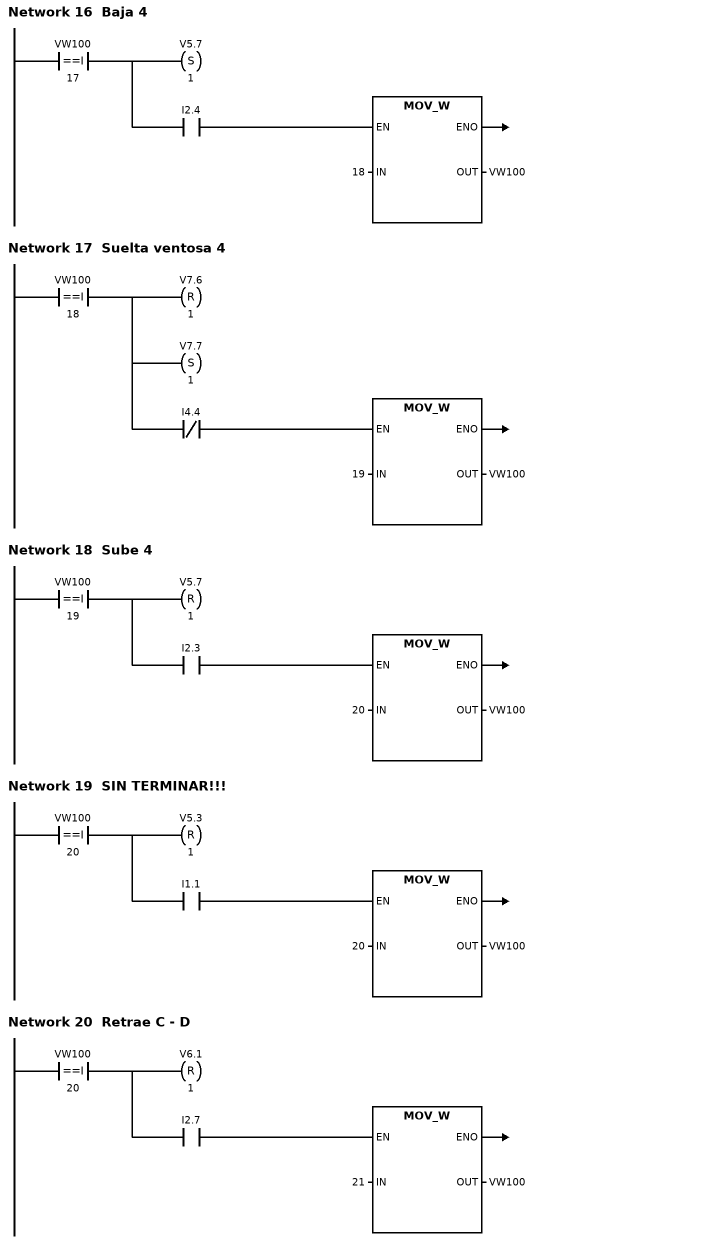
[picture p24: SBR1 networks 16-20]
Network 16 // Baja 4
LDW=   VW100, 17
S      V5.7, 1
A      I2.4
MOVW   18, VW100
Network 17 // Suelta ventosa 4
LDW=   VW100, 18
R      V7.6, 1
S      V7.7, 1
AN     I4.4
MOVW   19, VW100
Network 18 // Sube 4
LDW=   VW100, 19
R      V5.7, 1
A      I2.3
MOVW   20, VW100
Network 19 // SIN TERMINAR!!!
LDW=   VW100, 20
R      V5.3, 1
A      I1.1
MOVW   20, VW100
Network 20 // Retrae C - D
LDW=   VW100, 20
R      V6.1, 1
A      I2.7
MOVW   21, VW100
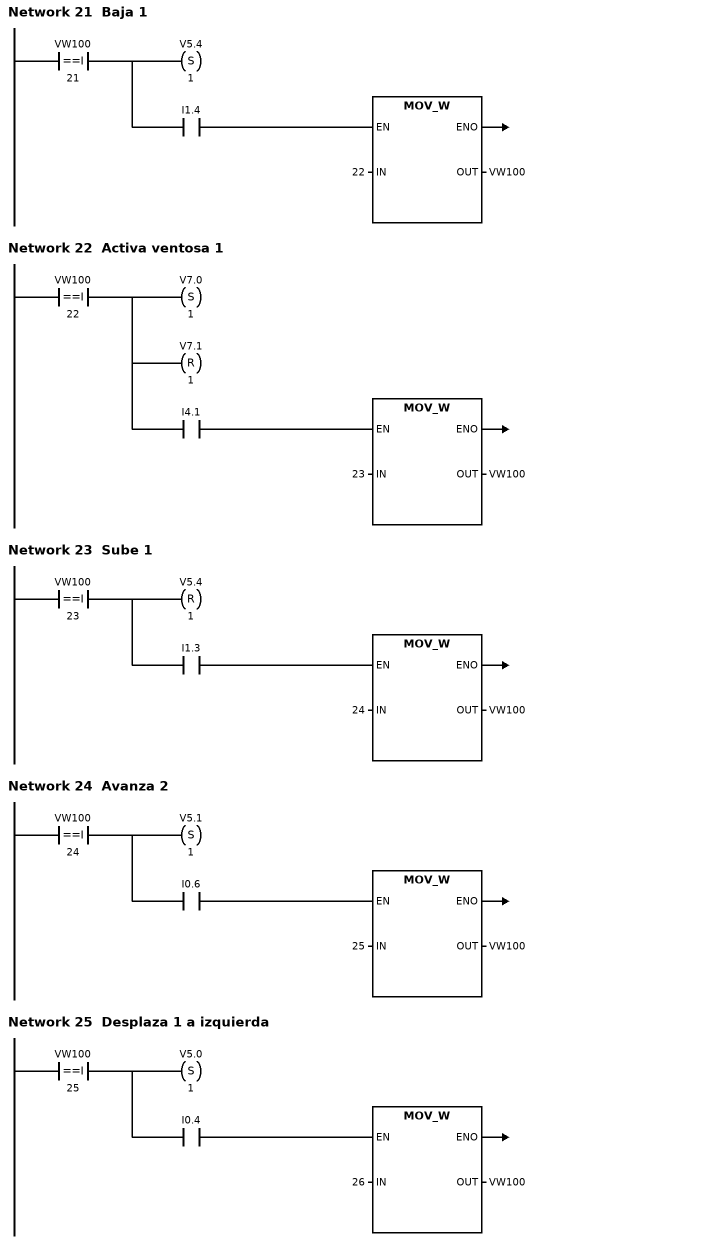
Network 21 // Baja 1
LDW=   VW100, 21
S      V5.4, 1
A      I1.4
MOVW   22, VW100
Network 22 // Activa ventosa 1
LDW=   VW100, 22
S      V7.0, 1
R      V7.1, 1
A      I4.1
MOVW   23, VW100
Network 23 // Sube 1
LDW=   VW100, 23
R      V5.4, 1
A      I1.3
MOVW   24, VW100
Network 24 // Avanza 2
LDW=   VW100, 24
S      V5.1, 1
A      I0.6
MOVW   25, VW100
Network 25 // Desplaza 1 a izquierda
LDW=   VW100, 25
S      V5.0, 1
A      I0.4
MOVW   26, VW100
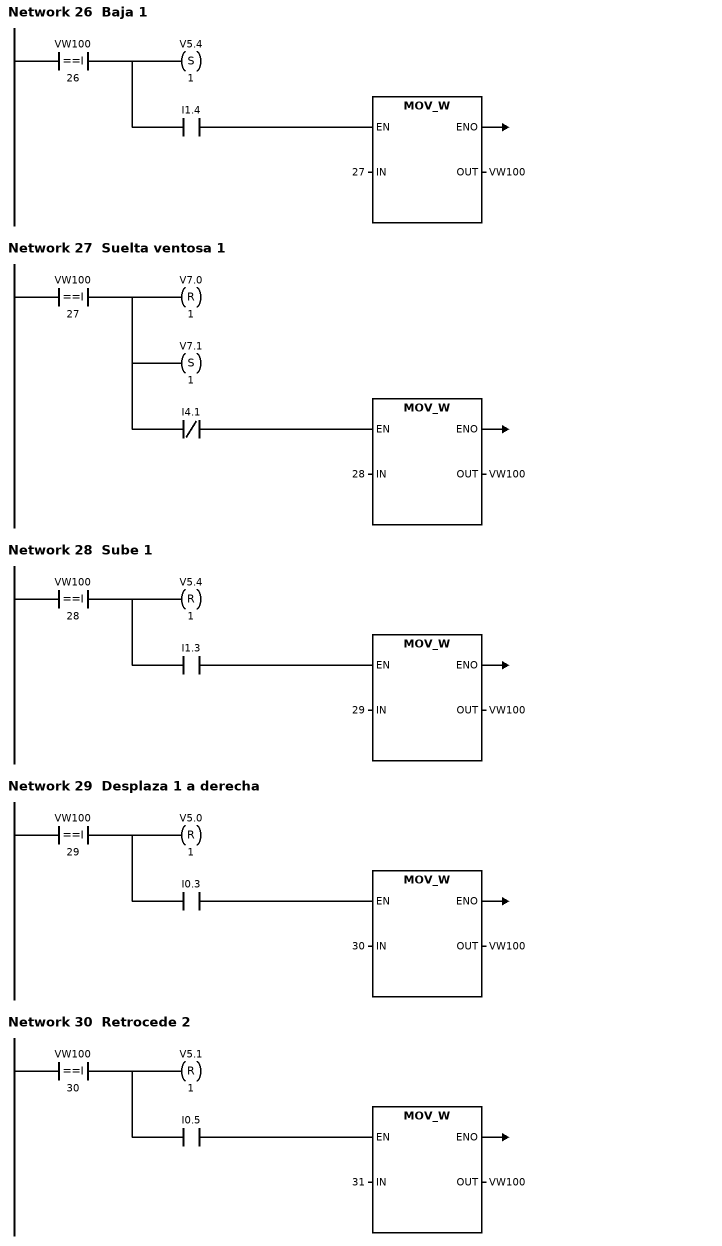
Network 26 // Baja 1
LDW=   VW100, 26
S      V5.4, 1
A      I1.4
MOVW   27, VW100
Network 27 // Suelta ventosa 1
LDW=   VW100, 27
R      V7.0, 1
S      V7.1, 1
AN     I4.1
MOVW   28, VW100
Network 28 // Sube 1
LDW=   VW100, 28
R      V5.4, 1
A      I1.3
MOVW   29, VW100
Network 29 // Desplaza 1 a derecha
LDW=   VW100, 29
R      V5.0, 1
A      I0.3
MOVW   30, VW100
Network 30 // Retrocede 2
LDW=   VW100, 30
R      V5.1, 1
A      I0.5
MOVW   31, VW100
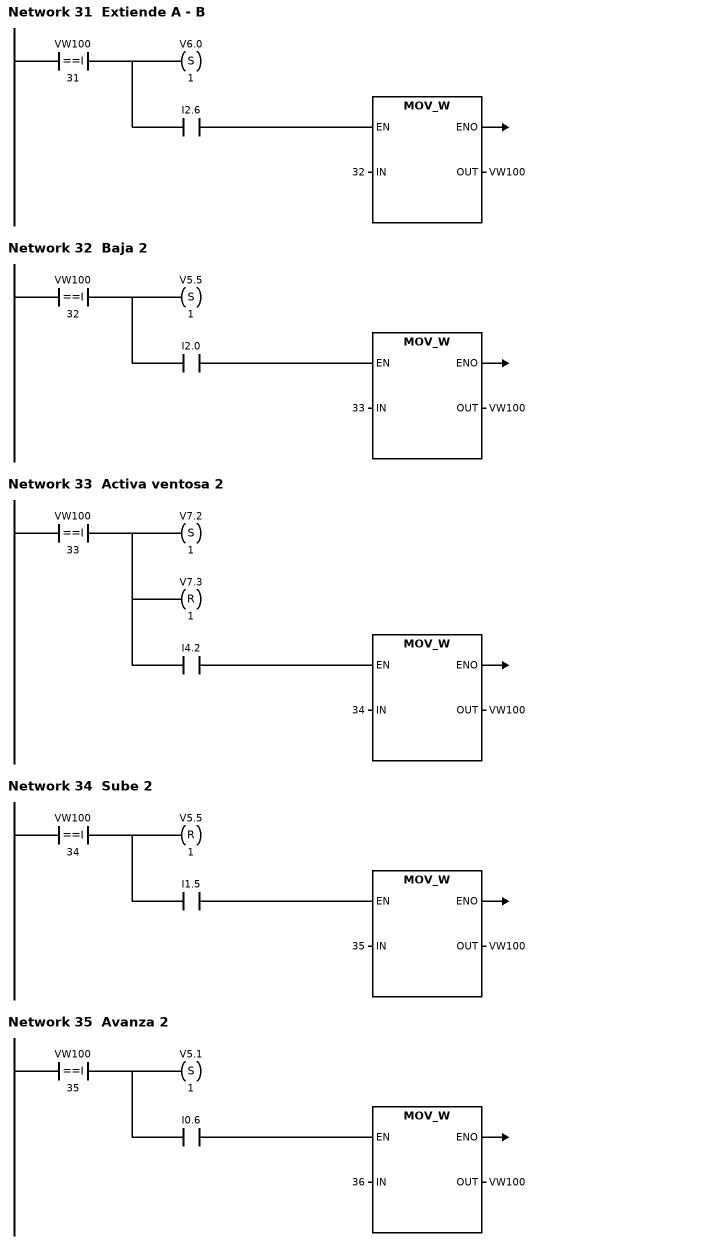
Network 31 // Extiende A - B
LDW=   VW100, 31
S      V6.0, 1
A      I2.6
MOVW   32, VW100
Network 32 // Baja 2
LDW=   VW100, 32
S      V5.5, 1
A      I2.0
MOVW   33, VW100
Network 33 // Activa ventosa 2
LDW=   VW100, 33
S      V7.2, 1
R      V7.3, 1
A      I4.2
MOVW   34, VW100
Network 34 // Sube 2
LDW=   VW100, 34
R      V5.5, 1
A      I1.5
MOVW   35, VW100
Network 35 // Avanza 2
LDW=   VW100, 35
S      V5.1, 1
A      I0.6
MOVW   36, VW100
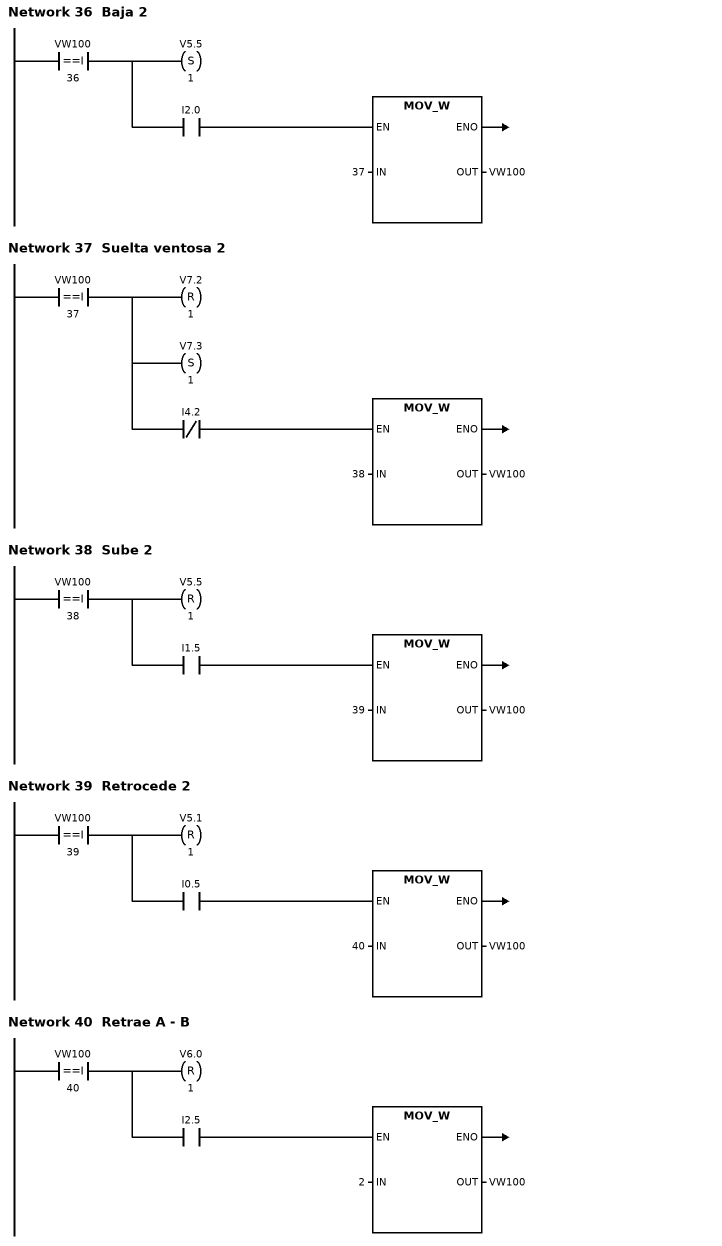
Network 36 // Baja 2
LDW=   VW100, 36
S      V5.5, 1
A      I2.0
MOVW   37, VW100
Network 37 // Suelta ventosa 2
LDW=   VW100, 37
R      V7.2, 1
S      V7.3, 1
AN     I4.2
MOVW   38, VW100
Network 38 // Sube 2
LDW=   VW100, 38
R      V5.5, 1
A      I1.5
MOVW   39, VW100
Network 39 // Retrocede 2
LDW=   VW100, 39
R      V5.1, 1
A      I0.5
MOVW   40, VW100
Network 40 // Retrae A - B
LDW=   VW100, 40
R      V6.0, 1
A      I2.5
MOVW   2, VW100
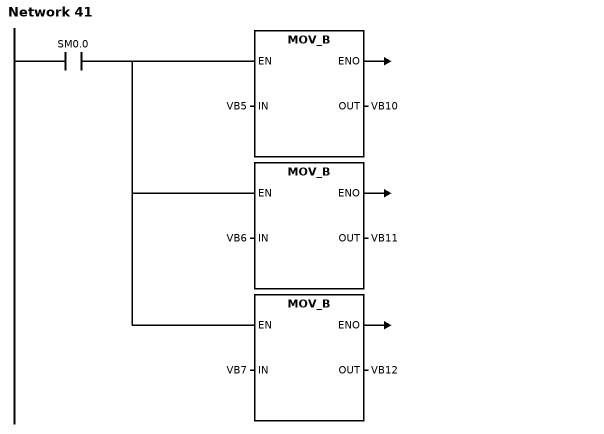
Network 41
LD     SM0.0
MOVB   VB5, VB10
MOVB   VB6, VB11
MOVB   VB7, VB12
END_SUBROUTINE_BLOCK

SUBROUTINE_BLOCK Control_salidas:SBR2
TITLE=COMENTARQOS DE LA SUBRUTQNA
BEGIN
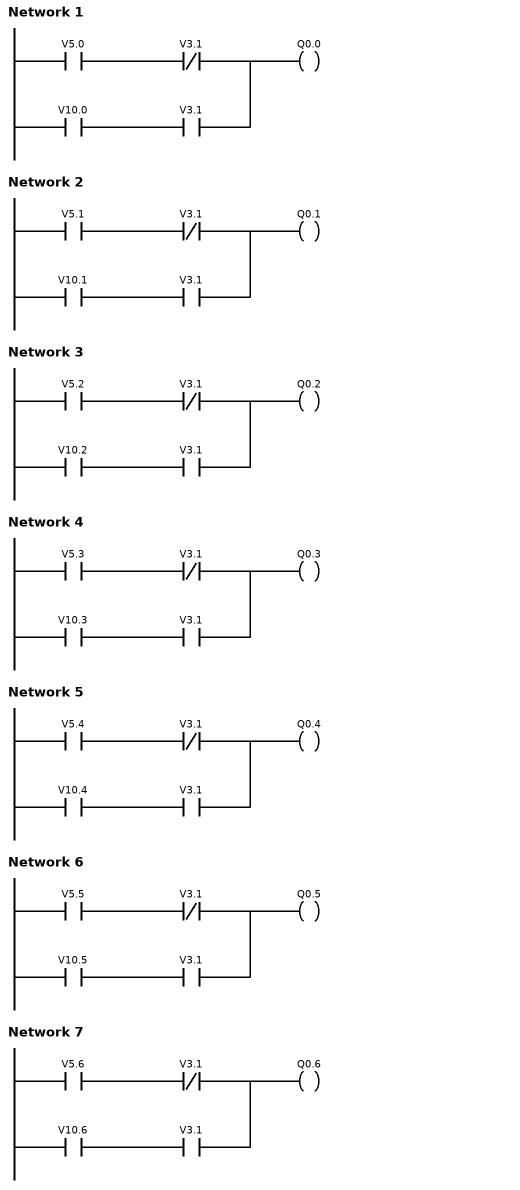
Network 1
LD     V5.0
AN     V3.1
LD     V10.0
A      V3.1
OLD
=      Q0.0
Network 2
LD     V5.1
AN     V3.1
LD     V10.1
A      V3.1
OLD
=      Q0.1
Network 3
LD     V5.2
AN     V3.1
LD     V10.2
A      V3.1
OLD
=      Q0.2
Network 4
LD     V5.3
AN     V3.1
LD     V10.3
A      V3.1
OLD
=      Q0.3
Network 5
LD     V5.4
AN     V3.1
LD     V10.4
A      V3.1
OLD
=      Q0.4
Network 6
LD     V5.5
AN     V3.1
LD     V10.5
A      V3.1
OLD
=      Q0.5
Network 7
LD     V5.6
AN     V3.1
LD     V10.6
A      V3.1
OLD
=      Q0.6
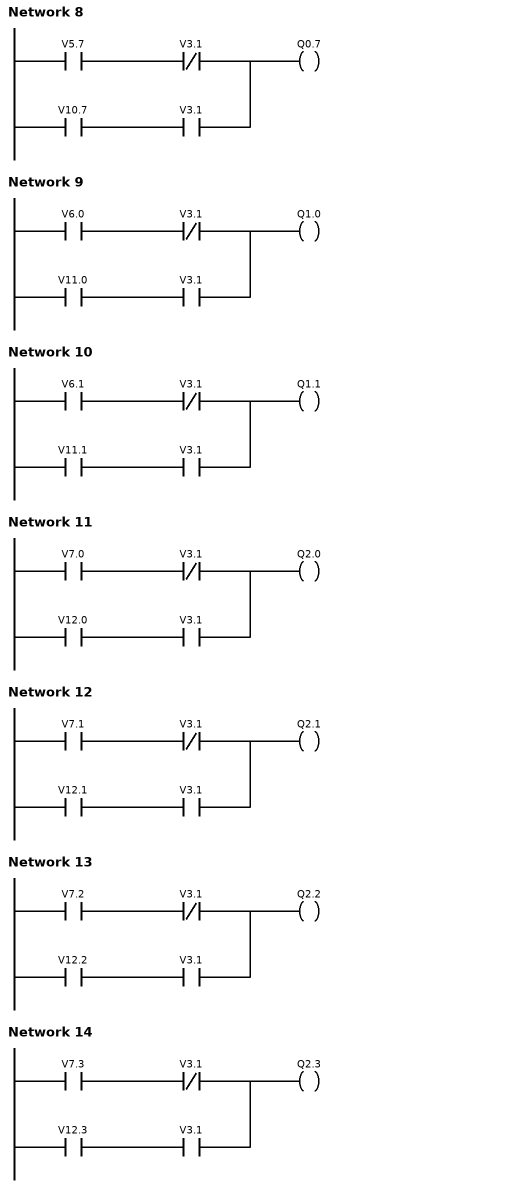
Network 8
LD     V5.7
AN     V3.1
LD     V10.7
A      V3.1
OLD
=      Q0.7
Network 9
LD     V6.0
AN     V3.1
LD     V11.0
A      V3.1
OLD
=      Q1.0
Network 10
LD     V6.1
AN     V3.1
LD     V11.1
A      V3.1
OLD
=      Q1.1
Network 11
LD     V7.0
AN     V3.1
LD     V12.0
A      V3.1
OLD
=      Q2.0
Network 12
LD     V7.1
AN     V3.1
LD     V12.1
A      V3.1
OLD
=      Q2.1
Network 13
LD     V7.2
AN     V3.1
LD     V12.2
A      V3.1
OLD
=      Q2.2
Network 14
LD     V7.3
AN     V3.1
LD     V12.3
A      V3.1
OLD
=      Q2.3
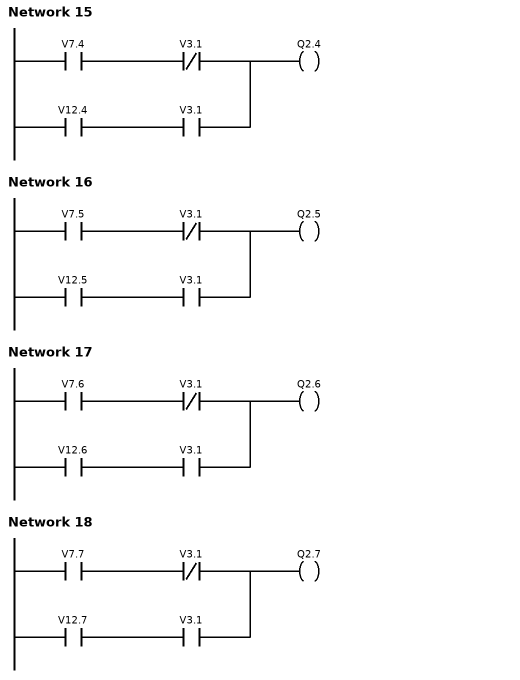
Network 15
LD     V7.4
AN     V3.1
LD     V12.4
A      V3.1
OLD
=      Q2.4
Network 16
LD     V7.5
AN     V3.1
LD     V12.5
A      V3.1
OLD
=      Q2.5
Network 17
LD     V7.6
AN     V3.1
LD     V12.6
A      V3.1
OLD
=      Q2.6
Network 18
LD     V7.7
AN     V3.1
LD     V12.7
A      V3.1
OLD
=      Q2.7
END_SUBROUTINE_BLOCK
